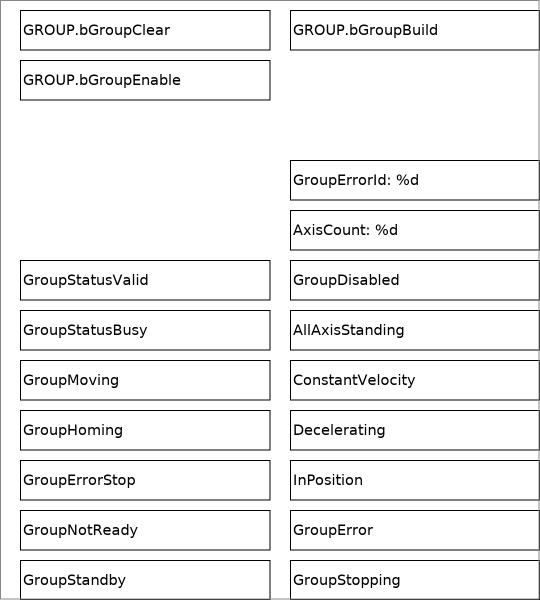
VISUALIZATION GROUP_VISU  // 540x600
    Rectangle (20,260 250x40), "GroupStatusValid", colour toggle: GVL_XTS.CaGroupInfo.GroupStatusValid
    Rectangle (20,310 250x40), "GroupStatusBusy", colour toggle: GVL_XTS.CaGroupInfo.GroupStatusBusy
    Rectangle (20,360 250x40), "GroupMoving", colour toggle: GVL_XTS.CaGroupInfo.GroupMoving
    Rectangle (20,410 250x40), "GroupHoming", colour toggle: GVL_XTS.CaGroupInfo.GroupHoming
    Rectangle (20,460 250x40), "GroupErrorStop", colour toggle: GVL_XTS.CaGroupInfo.GroupErrorStop
    Rectangle (20,510 250x40), "GroupNotReady", colour toggle: GVL_XTS.CaGroupInfo.GroupNotReady
    Rectangle (20,560 250x40), "GroupStandby", colour toggle: GVL_XTS.CaGroupInfo.GroupStandby
    Rectangle (290,560 250x40), "GroupStopping", colour toggle: GVL_XTS.CaGroupInfo.GroupStopping
    Rectangle (290,260 250x40), "GroupDisabled", colour toggle: GVL_XTS.CaGroupInfo.GroupDisabled
    Rectangle (290,310 250x40), "AllAxisStanding", colour toggle: GVL_XTS.CaGroupInfo.AllAxesStanding
    Rectangle (290,360 250x40), "ConstantVelocity", colour toggle: GVL_XTS.CaGroupInfo.ConstantVelocity
    Rectangle (290,410 250x40), "Decelerating", colour toggle: GVL_XTS.CaGroupInfo.Decelerating
    Rectangle (290,460 250x40), "InPosition", colour toggle: GVL_XTS.CaGroupInfo.InPosition
    Rectangle (290,510 250x40), "GroupError", colour toggle: GVL_XTS.CaGroupInfo.GroupError
    Rectangle (290,160 250x40), "GroupErrorId: %d", text variable: GVL_XTS.CaGroupInfo.GroupErrorId
    Rectangle (290,210 250x40), "AxisCount: %d", text variable: GVL_XTS.CaGroupInfo.AxisCount
    Rectangle (20,10 250x40), "GROUP.bGroupClear", colour toggle: GROUP.bGroupClear
        toggle GROUP.bGroupClear
    Rectangle (290,10 250x40), "GROUP.bGroupBuild", colour toggle: GROUP.bGroupBuild
        toggle GROUP.bGroupBuild
    Rectangle (20,60 250x40), "GROUP.bGroupEnable", colour toggle: GROUP.bGroupEnable
        toggle GROUP.bGroupEnable
END_VISUALIZATION

(* stored: Version 1.1.0.1, ProductVersion 3.1.4024.12
   Visu GROUP_VISU: Id {9dcaf819-5ca7-43b4-8101-6ccb4d5cb710} *)
